Staubli VAL3: StaubliSocket.dtx

mdesc mNomSpeed
sio sClient = {link=Socket\StlClient}
sio sServer = {link=Socket\StlServer}
